// Mitsubishi GX Works2 project: PLC01   PLC: Q02U

PROGRAM MAIN
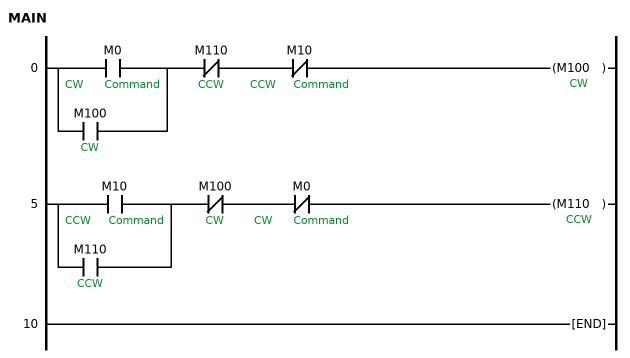
0     LD      M0  ; CW      Command
      OR      M100  ; CW
      ANI     M110  ; CCW
      ANI     M10  ; CCW     Command
      OUT     M100  ; CW
5     LD      M10  ; CCW     Command
      OR      M110  ; CCW
      ANI     M100  ; CW
      ANI     M0  ; CW      Command
      OUT     M110  ; CCW
10    END
END_PROGRAM

// device comments not shown above
M1  ; INTERLOCK
